FUNCTION_BLOCK FB_Window
VAR
    i : DINT; //loop counter
    SampleSpansBoxTime  : BOOL; //check if the data sample was an edge case between lines
    EnteredViaValidSide : BOOL; //TRUE if the line was a valid entry
    HasExitedBox        : BOOL; //TRUE if the line exited the box
    PermissionViolation : BOOL; // Flagged if it passes through an unpermitted line
    ValidEntrySide      : INT;  // 1 = Side A, 3 = Side C, 4 = Side D
    TrappedSuccessfully : BOOL; 
	
END_VAR
VAR_INPUT
	//data to check
	dataAxis: typeDataAxis;

    // Corner Points
    i1 : ST_BoxCorner; // Top-Left
    i2 : ST_BoxCorner; // Bottom-Left
    i3 : ST_BoxCorner; // Bottom-Right
    i4 : ST_BoxCorner; // Top-Right

    // Wall Permissions 
    PermSideA : ST_WallPermission; // Left Wall Permissions
    PermSideB : ST_WallPermission; // Right Wall Permissions
    PermSideC : ST_WallPermission; // Top Wall Permissions
    PermSideD : ST_WallPermission; // Bottom Wall Permissions
		
END_VAR

VAR_OUTPUT
    qPass : BOOL; // TRUE if data entered legally and followed all rules
    qFail : BOOL; // TRUE if any permission rule was violated or it leaked out
	qErrorCode : E_BoxResultCode; //diag codes
END_VAR

(*	^
	value (kN, etc)
	|
	|							C
	|			1_______________________________4
	|			|								|
	|			|								|
	|			|								|
	|			|			  /					|
	|			|			 /					|  
	|		A	|			/					|  B
	|			|		  /						|
	|			|	    /						|
	|			|	  /							|
	|-----------|----------------line-----------|-------
	|			|___/___________________________|
	|			2  /							3
	|			  /				D
	|		 	 /				
	|			/				
	----------------------------------------------------------------(grab)time->
	1	2	3	4	5	6	7	8	9 	10 	11	12	13	14	15	16	17 etc
	
	Each side of a box has a entry point, check which vector the data
	passes into
*)

// Reset tracking variables before running the historical loop
EnteredViaValidSide := FALSE;
HasExitedBox        := FALSE;
PermissionViolation := FALSE;
ValidEntrySide      := 0; 
qPass               := FALSE;
qFail               := FALSE;
qErrorCode          := E_BoxResultCode.Success; // Default to Success state

FOR i := 2 TO 20000 DO
    
    SampleSpansBoxTime := (dataAxis.grabTime[i] >= i2.PointXTime) AND (dataAxis.grabTime[i-1] <= i3.PointXTime);

    // =========================================================================
    // PART 1: ENTRY DETECTION & ENTRY PERMISSION CHECKS
    // =========================================================================
    IF NOT EnteredViaValidSide AND NOT PermissionViolation THEN
        
        // 1. SIDE A ENTRY (Left Wall)
        IF (dataAxis.grabTime[i-1] < i2.PointXTime) AND (dataAxis.grabTime[i] >= i2.PointXTime) THEN
            IF (dataAxis.grabData[i] > i2.PointYValue) AND (dataAxis.grabData[i] < i1.PointYValue) THEN
                
                IF PermSideA.IsNotPermittedToEnter OR NOT PermSideA.IsPermittedToEnter THEN
                    PermissionViolation := TRUE;
                    qErrorCode          := E_BoxResultCode.Err_IllegalEntry_SideA;
                ELSE
                    EnteredViaValidSide := TRUE;
                    ValidEntrySide      := 1; 
                END_IF
            END_IF
        END_IF

        // 2. SIDE D ENTRY (Bottom Wall)
        IF (dataAxis.grabTime[i] >= i2.PointXTime) AND (dataAxis.grabTime[i] <= i3.PointXTime) THEN
            IF (dataAxis.grabData[i-1] < i2.PointYValue) AND (dataAxis.grabData[i] >= i2.PointYValue) THEN
                
                IF PermSideD.IsNotPermittedToEnter OR NOT PermSideD.IsPermittedToEnter THEN
                    PermissionViolation := TRUE;
                    qErrorCode          := E_BoxResultCode.Err_IllegalEntry_SideD;
                ELSE
                    EnteredViaValidSide := TRUE;
                    ValidEntrySide      := 4; 
                END_IF
            END_IF
        END_IF
		
        // 3. SIDE C ENTRY (Top Wall)
        IF (dataAxis.grabTime[i] >= i2.PointXTime) AND (dataAxis.grabTime[i] <= i3.PointXTime) THEN
            IF (dataAxis.grabData[i-1] > i1.PointYValue) AND (dataAxis.grabData[i] <= i1.PointYValue) THEN
                
                IF PermSideC.IsNotPermittedToEnter OR NOT PermSideC.IsPermittedToEnter THEN
                    PermissionViolation := TRUE;
                    qErrorCode          := E_BoxResultCode.Err_IllegalEntry_SideC;
                ELSE
                    EnteredViaValidSide := TRUE;
                    ValidEntrySide      := 3; 
                END_IF
            END_IF
        END_IF
        
        // Break out instantly if the curve broke in through an illegal wall
        IF PermissionViolation THEN
            EXIT;
        END_IF
    END_IF

    // =========================================================================
    // PART 2: EXIT VIOLATION DETECTION (Evaluates immediately if Entered)
    // =========================================================================
    IF EnteredViaValidSide THEN 
        
        // 1. EXIT VIA SIDE B (Right Wall)
        IF (dataAxis.grabTime[i-1] <= i3.PointXTime) AND (dataAxis.grabTime[i] > i3.PointXTime) THEN
            IF (dataAxis.grabData[i] > i3.PointYValue) AND (dataAxis.grabData[i] < i4.PointYValue) THEN
                HasExitedBox := TRUE;
                IF PermSideB.IsNotPermittedToExit THEN
                    PermissionViolation := TRUE;
                    qErrorCode          := E_BoxResultCode.Violation_Exited_SideB;
                ELSE
                    qErrorCode          := E_BoxResultCode.Leak_Exited_SideB;
                END_IF
            END_IF
        END_IF

        // 2. EXIT VIA SIDE A (Left Wall)
        IF (dataAxis.grabTime[i-1] >= i2.PointXTime) AND (dataAxis.grabTime[i] < i2.PointXTime) THEN
            IF (dataAxis.grabData[i] > i2.PointYValue) AND (dataAxis.grabData[i] < i1.PointYValue) THEN
                HasExitedBox := TRUE;
                IF PermSideA.IsNotPermittedToExit THEN
                    PermissionViolation := TRUE;
                    qErrorCode          := E_BoxResultCode.Violation_Exited_SideA;
                ELSE
                    qErrorCode          := E_BoxResultCode.Leak_Exited_SideA;
                END_IF
            END_IF
        END_IF

        // 3. EXIT VIA SIDE C (Top Wall)
        IF SampleSpansBoxTime THEN
            IF (dataAxis.grabData[i-1] <= i1.PointYValue) AND (dataAxis.grabData[i] > i1.PointYValue) THEN
                HasExitedBox := TRUE;
                IF PermSideC.IsNotPermittedToExit THEN
                    PermissionViolation := TRUE;
                    qErrorCode          := E_BoxResultCode.Violation_Exited_SideC;
                ELSE
                    qErrorCode          := E_BoxResultCode.Leak_Exited_SideC;
                END_IF
            END_IF
        END_IF

        // 4. EXIT VIA SIDE D (Bottom Wall)
        IF SampleSpansBoxTime THEN
            IF (dataAxis.grabData[i-1] >= i2.PointYValue) AND (dataAxis.grabData[i] < i2.PointYValue) THEN
                HasExitedBox := TRUE;
                IF PermSideD.IsNotPermittedToExit THEN
                    PermissionViolation := TRUE;
                    qErrorCode          := E_BoxResultCode.Violation_Exited_SideD;
                ELSE
                    qErrorCode          := E_BoxResultCode.Leak_Exited_SideD;
                END_IF
            END_IF
        END_IF
        
        // Break loop early if an exit occurred or a specific permission rule was violated
        IF HasExitedBox OR PermissionViolation THEN
            EXIT; 
        END_IF

    END_IF

END_FOR

// =========================================================================
// PART 3: FINAL EVALUATION & MUTUALLY EXCLUSIVE OUTPUTS
// =========================================================================
// Catch the edge case where the loop finished but the signal never even hit a box boundary
IF NOT EnteredViaValidSide AND NOT PermissionViolation THEN
    qErrorCode := E_BoxResultCode.Err_NeverEnteredBox;
END_IF

// Evaluate final pass/fail flags
IF EnteredViaValidSide AND NOT HasExitedBox AND NOT PermissionViolation THEN
    qPass      := TRUE;
    qFail      := FALSE;
    qErrorCode := E_BoxResultCode.Success;
ELSE
    qPass      := FALSE;
    qFail      := TRUE;
END_IF

END_FUNCTION_BLOCK

(* stored: Version 1.1.0.1, ProductVersion 3.1.4024.11
   POU FB_Window: Id {4cf7a1dd-4be4-0676-17d1-6d8992ea43f1}, SpecialFunc None *)
